INTERFACE I_Linked_List

// Creates/Adds an node to the end of the list
METHOD Create
VAR_INPUT
	Data : T_DATA_TYPE; // Data to add to new node.
END_VAR
END_METHOD

// Empties/Clears/Deletes list
METHOD Empty
END_METHOD

METHOD FB_exit : BOOL
VAR_INPUT
	bInCopyCode : BOOL; // if TRUE, the exit method is called for exiting an instance that is copied afterwards (online change).
END_VAR
END_METHOD

METHOD FB_init : BOOL
VAR_INPUT
	bInitRetains : BOOL; // if TRUE, the retain variables are initialized (warm start / cold start)
	bInCopyCode : BOOL;  // if TRUE, the instance afterwards gets moved into the copy code (online change)
END_VAR
END_METHOD

// Inserts node at a specific position in the list
METHOD Insert
VAR_INPUT
	Data 		: T_DATA_TYPE; 	// Data to add to new node.
	nPosition 	: DINT;		// Position to add new node in list.
END_VAR
END_METHOD

// Checks of list is empty.
METHOD Is_Empty : BOOL
VAR_INPUT
END_VAR
END_METHOD

// Gets element at any position of the list, wuthout removing it.
METHOD Peek : T_DATA_TYPE
VAR_INPUT
	nPosition : DINT;
END_VAR
END_METHOD

// Deletes/pops a node at the front of the list 
METHOD Pop : T_DATA_TYPE
END_METHOD

// Adds/pushes a node at the front of the list 
METHOD Push
VAR_INPUT
		Data 	: T_DATA_TYPE;
END_VAR
END_METHOD

// Deletes node at a specific position in the list
METHOD Remove : T_DATA_TYPE
VAR_INPUT
	nPosition 	: DINT; // Position of node to delete.
END_VAR
END_METHOD

// Reverse list
METHOD Reverse
END_METHOD

// Searches list for the first instance of data and returns it's location and whether it's in the list.
METHOD Search : BOOL
VAR_INPUT
	Data : T_DATA_TYPE; // Data to find in list
END_VAR
VAR_OUTPUT
	nPosition : DINT; // Location of the data  starting from 0. -1 means data is not found in list
END_VAR
END_METHOD

// Traverse the list to display each node
METHOD Show
VAR_IN_OUT
	aList 		: ARRAY[*] OF T_DATA_TYPE; // Array to display data in list.
END_VAR
END_METHOD

// Gets size of the list
METHOD Size : DINT;
END_METHOD

END_INTERFACE

(* stored: Version 1.1.0.1, ProductVersion 3.1.4024.4
   Itf I_Linked_List: Id {9be330a0-0ade-448d-8db7-fb724b4527d2}
   Method Create: Id {2d5d8125-965d-48ee-93c7-5ae59a089256}
   Method Empty: Id {e4dbf123-31ce-45b7-8bfe-3c3176727c05}
   Method FB_exit: Id {530bc2ea-7812-493c-bb28-619b1117fab7}
   Method FB_init: Id {adbf37c6-d151-47b1-ab40-787bb853ece2}
   Method Insert: Id {cc99751b-2841-46ce-a15f-8c4f11f78e71}
   Method Is_Empty: Id {8b56dadb-dc80-42de-9e9a-516e804d4dd3}
   Method Peek: Id {66028890-0ba3-4fa9-ac10-bd31b89b344e}
   Method Pop: Id {9598b066-6092-4025-84fe-79e56beda60a}
   Method Push: Id {a3cd6a1f-bd78-45e9-8f76-1abc70bac56a}
   Method Remove: Id {1bc48630-7261-49e1-8543-62eb12c2b52c}
   Method Reverse: Id {d2b04faf-d1cd-4384-ba97-65ef9e7d26bf}
   Method Search: Id {02644848-c4d3-4937-bfda-fcb3bfd64cf9}
   Method Show: Id {b2cdbc30-559d-4e9f-a327-ce47d09791ed}
   Method Size: Id {e5340c3e-e4e4-41cc-9659-abfe315073eb} *)
